	rFlawWaterAfterAlcaliSet:=	arFlawWaterAfterAlcaliSet[4, wChosenRecipeLine4],
	rFlawWaterAfterAccidSet:=	arFlawWaterAfterAccidSet[4, wChosenRecipeLine4],
	rWaterAfterSterilFlaw:=	arWaterAfterSterilFlaw[4, wChosenRecipeLine4],
	rWaterAfterSterilConc:=	arWaterAfterSterilConc[4, wChosenRecipeLine4],
	rFlawWaterAfterAlcaliSet:=	arFlawWaterAfterAlcaliSet[4, wChosenRecipeLine4],
	rFlawWaterAfterAccidSet:=	arFlawWaterAfterAccidSet[4, wChosenRecipeLine4],
	wUsedWaterLevelOK:= wUsedWaterLevelOK,
	wUsedWaterLevelNotOK:= wUsedWaterLevelNotOK,
	wBackTget:= Heater_BackTget_4,
	xPause:= xPauseWashingLine4,
	xVoutOn:= xState_V411,
	xV_NotshortcutOn:= xState_V410,
	xV_UsedWaterInOn:= xState_V408,
	xV_AlkaliInOn:= xState_V406,
	xV_AccidInOn:= xState_V407,
	xV_WaterOutOn:= xState_V401,
	xV_UsedWaterOutOn:= xState_V402,
	xV_AlkaliOutOn:= xState_V404,
	xV_AccidOutOn:= xState_V403,
	xV_CycleOn:= xState_V405,
	xPumpOn:= Pump_OnAuto_4,
	rConcentration:= Conc_Line4,
	(*xAccidIsGoing:=xAccidIsGoing4,*)
	xFeedbackSwitch:= DI_FeedBackSwitchLine4,
	rWaterAfterSterilT:=arWaterAfterSterilT[4, wChosenRecipeLine4],
	wRecipeTimeRinse:= arWaterTime[4, wChosenRecipeLine4],
	wRecipeTimeAlcali:= arAlkaliTime[4, wChosenRecipeLine4],
	wRecipeTimeAccid:= arAccidTime[4, wChosenRecipeLine4],
	wAfterRinseConcAlk:= (*wAfterRinseConcAlk*)rConcSolutionStopoperationAlk,
	wAfterRinseConcAcc:= (*wAfterRinseConcAcc*)rConcSolutionStopoperationAcc,
	wAfterAlkWaterTime:= arAfterAlkaliWaterTime[4, wChosenRecipeLine4],
	wAfterAccWaterTime:= arAfterAccidWaterTime[4, wChosenRecipeLine4],
	rTwaterSet:= arTwaterSet[4, wChosenRecipeLine4],
	rTalcaliSet:= arTalkaliSet[4, wChosenRecipeLine4],
	rTaccidSet:= arTaccidSet[4, wChosenRecipeLine4],
	rConcAlcaliSet:=(* arConcAlkaliSet[4, wChosenRecipeLine4]*)rConcSolutionStartOperationAlk,
	rConcAccidSet:= (*arConcAccidSet[4, wChosenRecipeLine4]*)rConcSolutionStartOperationAcc,
	rFlawAlcaliSet:= arFlawAlkaliSet[4, wChosenRecipeLine4],
	rFlawWaterSet:= arFlawWaterSet[4, wChosenRecipeLine4],
	rFlawAccidSet:= arFlawAccidSet[4, wChosenRecipeLine4],
	wTsteril:= arTsterilSet[4, wChosenRecipeLine4],
	wFlawSteril:= arFlawSterilSet[4, wChosenRecipeLine4],
	rConcSteril:= arConcSterilSet[4, wChosenRecipeLine4],
	wSterilTime:= arSterilTime[4, wChosenRecipeLine4],
	wCountOfOperations:= 7,
	xStart:= xStartWashingLine4,
	xVout:= OnAuto_V411,
	xV_Notshortcut:= OnAuto_V410,
	xV_UsedWaterIn:= OnAuto_V408,
	xV_AlkaliIn:= OnAuto_V406,
	xV_AccidIn:= OnAuto_V407,
	xV_WaterOut:= OnAuto_V401,
	xV_UsedWaterOut:= OnAuto_V402,
	xV_AlkaliOut:= OnAuto_V404,
	xV_AccidOut:= OnAuto_V403,
	xV_Cycle:= OnAuto_V405,
	xV_Drainage:= OnAuto_V409,
	xPump:= Pump_OnAuto_4,
	xHeaterPower:= Heater_AutoSetT_4,
	xResetErrors:= xResetAlmAll,
	xPA:= PA_OnAuto_4,
	rToutSet:= Heater_AutoSetT_4,
	rFlawOutSet:= Pump_FlawAutoSet_4,
	xDone:=xWashingDone_Line4,
	State=> wWashingStateLine4,
	PauseState=> (*wWashingPauseStateLine4*),
	wTimePassed=> wWashingTimePassed4,
	wTimeOperationSet=> wWashingOperTimeSet4,
	wError=> wWashingErr_4);
END_IF
END_PROGRAM

(* POU VarsToOut, ST *)
PROGRAM VarsToOut
VAR

END_VAR
_DO_PumpOn_1:= DO_PumpOn_1;
(*
_DO_PumpOn_2:= DO_PumpOn_2;
_DO_PumpOn_3:= DO_PumpOn_3;
_DO_PumpOn_4:= DO_PumpOn_4;
 *)
_DO_PA11:= DO_PA11;
_DO_PA12:= DO_PA12;
_DO_PA1:= DO_PA1;
(*
_DO_PA2:= DO_PA2;
_DO_PA3:= DO_PA3;
_DO_PA4:= DO_PA4;
 *)
_DO_V110:= DO_V110;
(*
_DO_V210:= DO_V210;
_DO_V310:= DO_V310;
_DO_V410:= DO_V410;
*)
_DO_V111:= DO_V111;
(*
_DO_V211:= DO_V211;
_DO_V311:= DO_V311;
_DO_V411:= DO_V411;
*)
_DO_V101:= DO_V101;
_DO_V102:= DO_V102;
_DO_V103:= DO_V103;
_DO_V104:= DO_V104;
_DO_V105:= DO_V105;
_DO_V106:= DO_V106;
_DO_V107:= DO_V107;
_DO_V108:= DO_V108;
_DO_V109:= DO_V109;
(*
_DO_V201:= DO_V201;
_DO_V202:= DO_V202;
_DO_V203:= DO_V203;
_DO_V204:= DO_V204;
_DO_V205:= DO_V205;
_DO_V206:= DO_V206;
_DO_V207:= DO_V207;
_DO_V208:= DO_V208;
_DO_V209:= DO_V209;
_DO_V301:= DO_V301;
_DO_V302:= DO_V302;
_DO_V303:= DO_V303;
_DO_V304:= DO_V304;
_DO_V305:= DO_V305;
_DO_V306:= DO_V306;
_DO_V307:= DO_V307;
_DO_V308:= DO_V308;
_DO_V309:= DO_V309;
_DO_V401:= DO_V401;
_DO_V402:= DO_V402;
_DO_V403:= DO_V403;
_DO_V404:= DO_V404;
_DO_V405:= DO_V405;
_DO_V406:= DO_V406;
_DO_V407:= DO_V407;
_DO_V408:= DO_V408;
_DO_V409:= DO_V409;
 
_DO_V501:= DO_V501;

_DO_V511:= DO_V511;
_DO_V510:= DO_V510;
_DO_V512:= DO_V512;
_DO_V513:= DO_V513;
_DO_V514:= DO_V514;
_DO_V515:= DO_V515;


_SwitchOnRemotePump_1	:=	SwitchOnRemotePump_1	;
_SwitchOnRemotePump_2	:=	SwitchOnRemotePump_2	;
_SwitchOnRemotePump_3	:=	SwitchOnRemotePump_3	;
_SwitchOnRemotePump_4	:=	SwitchOnRemotePump_4	;


_Ready_Line_2 :=SwitchOnRemotePump_1_2;
_Working_Line_2 :=SwitchOnRemotePump_1_1;
_Working_Pump_2:=SwitchOnRemotePump_1_3;


_AO_PumpSpeedSet_1:= AO_PumpSpeedSet_1;
_AO_PumpSpeedSet_2:= AO_PumpSpeedSet_2;
_AO_PumpSpeedSet_3:= AO_PumpSpeedSet_3;
_AO_PumpSpeedSet_4:= AO_PumpSpeedSet_4;
 *)
_AO_HeaterPowerSet_1:= AO_HeaterPowerSet_1;
(*
_AO_HeaterPowerSet_2:= AO_HeaterPowerSet_2;
_AO_HeaterPowerSet_3:= AO_HeaterPowerSet_3;
_AO_HeaterPowerSet_4:= AO_HeaterPowerSet_4;
*)
END_PROGRAM

(* POU Device/Sensors/fb_counter, ST *)
FUNCTION_BLOCK fb_counter
VAR_INPUT
	repair	:					BOOL	;
	counter	:				BOOL	;
	counter_valueStep	:	REAL	:=	1.0	;
	counter_init_value	:	REAL	;		
	start	:					BOOL	;
END_VAR

VAR_IN_OUT
	reset:			BOOL;
END_VAR

VAR_OUTPUT
	result:						REAL;
END_VAR

VAR
	status_counter:		BOOL;
END_VAR
(*couter di signals*)
IF repair = FALSE
  THEN
    IF start = TRUE
      THEN
        IF status_counter <> counter
          THEN
            IF counter = TRUE
              THEN
                result:= result + counter_valueStep;
            END_IF;
        END_IF;
        status_counter := counter;
    END_IF;

    IF reset = TRUE
      THEN
        reset:= FALSE;
        result:= counter_init_value;
    END_IF;
  ELSE
    result:= 0;
    reset:=FALSE;
    status_counter:= FALSE;
END_IF;
END_FUNCTION_BLOCK

(* POU Device/Sensors/fb_crash_to_int, ST *)
FUNCTION_BLOCK fb_crash_to_int
VAR_INPUT
	repair	:	BOOL	;
	crash_1	:	BOOL	;
	crash_2	:	BOOL	;
	crash_3	:	BOOL	;
	crash_4	:	BOOL	;
	crash_5	:	BOOL	;
	crash_6	:	BOOL	;
	crash_7	:	BOOL	;
	crash_8	:	BOOL	;
	crash_9	:	BOOL	;
	crash_10	:	BOOL	;

END_VAR
VAR_OUTPUT
	rezult_int_crash:	WORD;
END_VAR
VAR
END_VAR
IF repair = FALSE
  THEN
    rezult_int_crash:= INT_TO_WORD(
      (1) * BOOL_TO_INT(crash_1 OR crash_2 OR crash_3 OR crash_4 OR crash_5 OR crash_6 OR crash_7 OR crash_8 OR crash_9 OR crash_10) +
      (2) * BOOL_TO_INT(crash_1) +
      (4) * BOOL_TO_INT(crash_2) +
      (8) * BOOL_TO_INT(crash_3) +
      (16) * BOOL_TO_INT(crash_4) +
      (32) * BOOL_TO_INT(crash_5) +
      (64) * BOOL_TO_INT(crash_6) +
      (128) * BOOL_TO_INT(crash_7) +
      (256) * BOOL_TO_INT(crash_8) +
      (512) * BOOL_TO_INT(crash_9) +
      (1024) * BOOL_TO_INT(crash_10) );
  ELSE
      rezult_int_crash:= 0;
END_IF;
END_FUNCTION_BLOCK

(* POU _ExtraFB/ControlFB/fb_digout_signal, ST *)
FUNCTION_BLOCK fb_digout_signal
VAR_INPUT
	repair	:						BOOL	;
	out_signal_for_repair	:		BOOL	;
	use_smoothing	:			BOOL	;
	time_wait	:					TIME	:=	T#1s500ms	;
	input	:						BOOL	;

END_VAR
VAR_OUTPUT
	digout:							BOOL;
END_VAR
VAR
	perem_input:					BOOL	;
	TON_wait:						TON;
END_VAR
IF repair = FALSE
  THEN
    IF use_smoothing = FALSE
      THEN
        (*???? ?????? ??????????? ????? ?????*)
        digout:= input;
      ELSE
        (*???? ???? ???????? ??????? ?????? ? ?? ?????? ?????????????? ???????? ????????*)
        IF input <> perem_input
          THEN
            TON_wait( IN:=TRUE, PT:= time_wait);
          ELSE
            TON_wait( IN:=FALSE, PT:= time_wait);
        END_IF;
        IF TON_wait.Q = TRUE
          THEN
            digout:= input;
            perem_input:= input;
            TON_wait( IN:=FALSE, PT:= time_wait);
        END_IF;
    END_IF;
  ELSE
    digout:= out_signal_for_repair;
END_IF;
  
END_FUNCTION_BLOCK

(* POU Device/Sensors/fb_speed_di, ST *)
FUNCTION_BLOCK fb_speed_di
VAR_INPUT
	repair	:				BOOL	;
	di_speed	:			BOOL	;
	real_obor_min	:	REAL	:=	1500.0	;
	max_speed	:		REAL	:=	1500.0	;
	time_update	:		DINT	:=	1500	;

END_VAR
VAR_OUTPUT
	result_speed:			REAL;
END_VAR
VAR
	TON_speed	:		TON	;
	status_di_speed	:	BOOL	;
	count_impuls	:		REAL	;

END_VAR
(*translate di speed in speed*)
IF repair = FALSE
  THEN
    IF (status_di_speed = FALSE AND di_speed = TRUE)
      THEN
        count_impuls:= count_impuls + 1;
    END_IF;

    TON_speed( IN:= TRUE, PT:=  DINT_TO_TIME(time_update));
    IF TON_speed.Q = TRUE
      THEN
        TON_speed( IN:= FALSE, PT:=  t#60s);
        IF real_obor_min <> 0 AND time_update <> 0
          THEN
            result_speed:= max_speed * ((count_impuls * 60.0 / (DINT_TO_REAL(time_update) / 1000.0)) / real_obor_min);
          ELSE
            result_speed:= 0;
        END_IF;
        count_impuls:= 0;
    END_IF;

    status_di_speed:= di_speed;
  ELSE
    result_speed:= 0;
    TON_speed( IN:= FALSE, PT:=  t#10d);
    status_di_speed:= FALSE;
    count_impuls:= 0;
END_IF;
END_FUNCTION_BLOCK

(* POU Device/Sensors/fb_tank, ST *)
FUNCTION_BLOCK fb_tank
VAR_INPUT
	use_smoothing	:	BOOL	;
	time_wait	:			TIME	:=	T#1s500ms	;
	input_H	:			BOOL	;
	input_M	:			BOOL	;
	input_L	:			BOOL	;

END_VAR
VAR_OUTPUT
	result_H	:			BOOL	;
	result_M	:			BOOL	;
	result_L	:			BOOL	;
	crash_value	:		BOOL	;
	out_crash_int	:		WORD	;

END_VAR
VAR
	sensor_H	:			fb_digout_signal	;
	sensor_M	:			fb_digout_signal	;
	sensor_L	:			fb_digout_signal	;
	db_crash_to_int	:	fb_crash_to_int	;

END_VAR
(*high level*)
sensor_H(
  repair:=                 FALSE,
  out_signal_for_repair:=  FALSE,
  use_smoothing:=          use_smoothing,
  time_wait:=              time_wait,
  input:=                  input_H,
  digout=>                 result_H);
(*middle level*)
sensor_M(
  repair:=                 FALSE,
  out_signal_for_repair:=  FALSE,
  use_smoothing:=          use_smoothing,
  time_wait:=              time_wait,
  input:=                  input_M,
  digout=>                 result_M);
(*lower level*)
sensor_L(
  repair:=                 FALSE,
  out_signal_for_repair:=  FALSE,
  use_smoothing:=          use_smoothing,
  time_wait:=              time_wait,
  input:=                  input_L,
  digout=>                 result_L);

(*IF (result_M = TRUE AND result_L = FALSE) OR (result_H = TRUE AND result_M = FALSE)
  THEN
    crash_value:= TRUE;
  ELSE
    crash_value:= FALSE;
END_IF;*)
    crash_value:= FALSE;

  
(*?????? ??? ??????*)
db_crash_to_int(
  crash_1:= crash_value );
out_crash_int:= db_crash_to_int.rezult_int_crash;
END_FUNCTION_BLOCK

(* POU Process/SelfWashing/fbWashingTanks, ST *)
FUNCTION_BLOCK fbWashingTanks
VAR_INPUT
	xV_AllInState:					BOOL;
	xV_DrainageState:			BOOL;
	xV_TankInState:				BOOL;
	xV_CleanerOutState:			BOOL;
	xV_PrevCleanerOutState:		BOOL;
	wOperTimeSet:				WORD;
	NextState:							SelfWashingStates;
END_VAR
VAR_IN_OUT

	xV_AllIn:						BOOL;
	xV_Drainage:					BOOL;
	xV_TankIn:						BOOL;
	xV_CleanerOut:				BOOL;
	xV_PrevCleanerOut:			BOOL;
	xPumpOn:						BOOL;
	State:							SelfWashingStates;
END_VAR
VAR_OUTPUT
END_VAR
VAR
	tnWashing:					TON;
	xStartOper:					BOOL;
END_VAR
xV_AllIn:=				TRUE;
xV_Drainage:=		TRUE;
xV_TankIn:=			TRUE;
xV_CleanerOut:=		TRUE;
xV_PrevCleanerOut:=	FALSE;

IF (NOT xV_PrevCleanerOutState) AND xV_AllInState AND xV_DrainageState AND xV_TankInState AND xV_CleanerOutState THEN
	xPumpOn:=TRUE;
	xStartOper:=TRUE;
END_IF

tnWashing(IN:=xStartOper,  PT:= (WORD_TO_TIME(wOperTimeSet))*1000);
IF tnWashing.Q THEN
	tnWashing(IN:=FALSE);
	xStartOper:=FALSE;
	State:= NextState;
END_IF
END_FUNCTION_BLOCK

(* POU Device/Sensors/fnAI_TO_CURRENCY, ST *)
FUNCTION fnAI_TO_CURRENCY : REAL
VAR_INPUT
	AI:	WORD;
END_VAR
VAR
	result:REAL;
END_VAR
result:=(WORD_TO_REAL(AI)/32762)*20;
fnAI_TO_CURRENCY:=result;
END_FUNCTION

(* POU Device/Sensors/fnPressureToVolume, ST *)
FUNCTION fnPressureToVolume : REAL
VAR_INPUT
	Pressure:	REAL;
	Square:	REAL;
END_VAR
VAR
END_VAR
fnPressureToVolume:=(Pressure*Square)/9.79038;
END_FUNCTION
